PROGRAM prgMisc
VAR	
	H31_SRBVH3_RADH3_TR_RG_extSetpointActive		: INT;											//{#lynus.ag#()}
	H31_SRBVH3_RADH3_TR_RGextSetpointActiveB 	: BOOL;											//{#lynus.ag#()}
	m_Enable_HeartBeat								: BOOL;											//{#lynus.ag#()}
	ton_Delay: Ton;
END_VAR

IF m_Enable_HeartBeat AND ton_Delay.Q THEN
	H31_SRBVH3_RADH3_TR_RG_extSetpointActive := 1;
	H31_SRBVH3_RADH3_TR_RGextSetpointActiveB := TRUE;
ELSIF NOT m_Enable_HeartBeat AND ton_Delay.Q THEN
	H31_SRBVH3_RADH3_TR_RG_extSetpointActive := 0;	
	H31_SRBVH3_RADH3_TR_RGextSetpointActiveB := FALSE;
END_IF

ton_Delay(In:= NOT ton_Delay.Q, PT := T#60S);

END_PROGRAM

(* stored: Version 1.1.0.1, ProductVersion 3.1.4024.12
   POU prgMisc: Id {dd7dc983-641c-4b2a-8dec-aa875cb99a53}, SpecialFunc None *)
